(* IEC 61131-3 sources: skladplc/, 9 files *)

(* ---- prgMaindomaci.ST ---- *)
VAR_GLOBAL
cidloAnalog0 at %XW34:int;
cidloAnalog1 at %XW46:int;
cidlo_horiz at %X100.4:bool;
cidlo_verti at %X100.7:bool;
cidlo_rameno_zadni at %X10.7:bool;
doprav_cidlo_zad at %X100.6:bool;
doprav_cidlo_pre at %X100.5:bool;
zk0 at %X101.0:bool;
zk1 at %X101.1:bool;
zk2 at %X101.2:bool;
zk3 at %X101.3:bool;
doprav_do at %Y32.4:bool;//dopravnik, dovnitr
doprav_ve at %Y32.5:bool;//dopravnik, ven
horiz_vl at %Y32.6:bool;//horizontalni, vlevo:ccw
horiz_vp at %Y32.7:bool;//horizontalni, vpravo:cw
verti_do at %Y33.0:bool;//vertikalni, dolu
verti_na at %Y33.1:bool;//vertikalni, nahoru
ram_vy at %Y33.2:bool;//rameno, vysun
ram_vs at %Y33.3:bool;//rameno, vsun
horiz_ink:udint;
verti_ink:udint;
cas at %S13.2:bool;
kalibruj:bool:=0;
misto:bool:=0;

pomoc, pomoc1:bool;

casovac, casovac1, casovac2:TON;
(*
PolohaVerti: array[0..4] of udint :=[3852,1892,204,3420];
PolohaHoriz: array[0..4] of udint:=[9403,6462,3629,12];
Obsazenost: array [0..9] of int:=[0,0,0,0,0,0,0,0,0,0]; //not completed
*)
bar:int;
umistit:bool:=0;
nalozeno:bool:=0;
pozice0:int:=0;
pozice1:int:=0;
pozice2:int:=0;

END_VAR
FUNCTION manualni:bool     //HOTOVO, funkce pro servisni ovladani jednotky, pozdeji se smaze
   horiz_vp:=zk0 and not zk3;
   verti_na:=zk1 and not zk3;
   ram_vs:=zk2 and not zk3;
   horiz_vl:=zk0 and  zk3;
   verti_do:=zk1 and  zk3;
   ram_vy:=zk2 and  zk3;
END_FUNCTION
FUNCTION kalibrace:bool  //HOTOVO, funkce na uvodni kalibraci jednotky
   IF not cidlo_rameno_zadni then;
      ram_vs:=1;
      else ram_vs:=0;
      IF not cidlo_horiz then;
         horiz_vp:=1;
         else horiz_vp:=0;
      END_IF;
      IF not cidlo_verti then;
         verti_na:=1;
         else verti_na:=0;
      END_IF;
   END_IF;
   IF cidlo_rameno_zadni AND cidlo_horiz AND cidlo_verti then;
      kalibrace:=1;
   END_IF;
END_FUNCTION

FUNCTION umisti:bool
   IF cidloAnalog0<cidloAnalog1 then;
      IF verti_ink < 1892 then;
         verti_do:=1;
      ELSE
         verti_do:=0;
      END_IF;
      IF horiz_ink < 6462 then;
         horiz_vl:=1;
      ELSE
         horiz_vl:=0;
      END_IF;
      Obsazenost[pozice1]:=1;

      //
   ELSIF (cidloAnalog0<3600 AND cidloAnalog1<3600) then;
      IF verti_ink < 3852 then;
         verti_do:=1;
      ELSE
         verti_do:=0;
      END_IF;
      IF horiz_ink < 9403 then;
         horiz_vl:=1;
      ELSE
         horiz_vl:=0;
      END_IF;
      Obsazenost[pozice0]:=1;

      //
   ELSIF cidloAnalog0>cidloAnalog1  then;  //
      IF verti_ink < 204 then;
         verti_do:=1;
      ELSE
         verti_do:=0;
      END_IF;
      IF horiz_ink < 3629 then;
         horiz_vl:=1;
      ELSE
         horiz_vl:=0;
      END_IF;
      Obsazenost[pozice2]:=1;

      //
   END_IF;
END_FUNCTION
FUNCTION nakladani:bool //funkce pro posun dopravniku s obrokem do nakladaci oblasti
   IF verti_ink < 3350 then; //dojede na vertikalni polohu nakladaci oblasti
      verti_do:=1;
   ELSE
      verti_do:=0;
      pomoc1:=1;
   END_IF;
   IF horiz_ink < 10 then; //dojede na horizontalni polohu nakladaci oblasti
      horiz_vl:=1;
   ELSE
      horiz_vl:=0;
   END_IF;
   IF pomoc1 and not casovac1.Q then; //pokud je ve vertikalni poloze oblasti, zacne na 3s vysouvat rameno = paleta se posadi na dopravnik v nakl. obasti
      ram_vy:=1;
      casovac1(IN:=1, PT:=T#3s); //misto jednicky promenna - nulovani
   ELSIF nalozeno and casovac1.Q then; //pokud uzivatel stiskne tlacitko, ze barevny obrok vlozil, tak se paleta vrati zpet na rameno a to se zatahne
      doprav_
      ram_vy:=0;
      casovac2(IN:1, PT:=T#3s);
      ram_vs:=ram_vs and casovac2.Q
   END_IF;
END_FUNCTION
FUNCTION barva:int //funkce pro určení barvy + vypsání požadované barvy obroku na displej PLC
//hodnota 31500 pro analogove cidlo znamena, ze na dane pozici je cerna barva = neni bily prouzek
   IF not doprav_cidlo_pre AND doprav_cidlo_zad then;
      doprav_do:=1;

      barva:=-1;
      IF (cidloAnalog0=31500 AND cidloAnalog0>cidloAnalog1) then; //bily obrok, nahore bila
        //vypsat na displej BILA

      ELSIF (cidloAnalog1=31500 AND cidloAnalog0<cidloAnalog1) then; //cerveny obrok, dole bila
        //vypsat na displej CERVENA

      ELSIF (cidloAnalog0=31500 AND cidloAnalog0=cidloAnalog1) then; //modry obrok, nikde bila
        //vypsat na displej MODRA

      END_IF;

   END_IF;
   doprav_do:=doprav_cidlo_zad AND doprav_do;

END_FUNCTION
FUNCTION hybej:bool //funkce, ktera podle definovani barvy z funkce barva() urci na jakou pozici se ma naplnena paleta umistit v regalu
   IF not doprav_cidlo_pre AND doprav_cidlo_zad then;
      doprav_do:=1;
      //sken barvy
      IF (umistit) then;
         IF not doprav_cidlo_zad then; //zajisti, ze dopravnik prestane presouvat prazdnou paletu do zadni oblasti jakmile do ni dorazi
            doprav_do:=1;
            doprav_ve:=doprav_cidlo_pre AND doprav_ve;
            nakladej:=nakladani();
            IF nakladej then;
               umisti();
            END_IF;
         END_IF;
         IF (barva() = 0) then;

         ELSIF (barva() = 1) then;S

         ELSIF (barva () = 2) then;

         END_IF;
      END_IF;
      //ceka na potvrzeni vlozeni - stisk tlacitka
   END_IF;

   doprav_do:=doprav_cidlo_zad AND doprav_do;
END_FUNCTION

PROGRAM prgMain
VAR
   cidlo0, cidlo1:INT;
   pomoc:bool;
END_VAR
horiz_ink:=inkrementalni_horiz;
verti_ink:=inkrementalni_verti;
pomoc:=0;
cidlo0:=cidloAnalog0;
cidlo1:=cidloAnalog1;
IF not kalibruj then;     //uvodni kalibrace a pak uvolni system pro dalsi pouziti
   kalibruj:=kalibrace(); //funkce na uvodni kalibraci jednotky
ELSE
   IF casovac.Q then;
      ridSlovo:=1;
      ridSlovo1:=1;
      pomoc:=1;
      //manualni();
      //hybej();
      barva();
   ELSE
      ridSlovo:=2;
      ridSlovo1:=2;
      casovac(IN:=1, PT:=T#1s);
   END_IF;
END_IF;
END_PROGRAM

(* ---- ridici().ST ---- *)
VAR_GLOBAL
   horizontal:int:=0;
   vertikal:int:=0;
   blokace:bool:=0;
END_VAR
FUNCTION ridici:bool
   IF not blokace then
      IF not nabirani.probehlo then
         nabirani(i:=vertikal, j:=horizontal);
      ELSE
         IF not hybej.odvezl then
            hybej();
         ELSE
            IF not vraceni.vraceno then
               //hlavni_barva:=3;
               vraceni(i:=vertikal, j:=horizontal);
            ELSE
               IF horizontal<2 then //podminka pro posun v polich
                  horizontal:=horizontal+1; //posun v horizontalnim poli
                  nabirani.probehlo:=0;
                  hybej.odvezl:=0;
                  vraceni.vraceno:=0;
               END_IF;
               IF horizontal=2 AND vraceni.vraceno then
                  IF vertikal<2 then
                     vertikal:=vertikal+1;
                     horizontal:=-1;
                  ELSE
                     blokace:=1;
                  END_IF;
               END_IF;
            END_IF;
         END_IF;
      END_IF;
   ELSE
      kalibrace();
   END_IF;
END_FUNCTION

(* ---- kalibrace().ST ---- *)
FUNCTION kalibrace:bool //funkce na kalibraci jednotky
   IF not cidlo_rameno_zad then //zatahne rameno
      ram_vs:=1;
   ELSE
      ram_vs:=0;
      IF not cidlo_horiz then //narazi na horizontalni snimac
         horiz_vp:=1;
      ELSE
         horiz_vp:=0;
      END_IF;
      IF not cidlo_verti then //narazi na vertikalni snimac
         verti_na:=1;
      ELSE
         verti_na:=0;
      END_IF;
   END_IF;
   IF cidlo_rameno_zad AND cidlo_horiz AND cidlo_verti then //"vrati", ze probehla funkce
      kalibrace:=1;
   END_IF;
END_FUNCTION

(* ---- nakladani().st ---- *)
FUNCTION nakladani:bool //funkce pro posun jiz nalozene prazdne palety do dopravnikove oblasti + odebrani naplnene palety
   VAR
      verti:udint:=verti_ink;
      horiz:udint:=horiz_ink;
      pomoc:bool:=0;
      pomoc1:bool:=0;
   END_VAR
   IF verti < 3250 then; //dojede na vertikalni polohu nakladaci oblasti
      verti_do:=1;
   ELSIF verti > 3250 then;
      verti_na:=1;
   ELSE
      verti_do:=0;
      verti_na:=0;
      pomoc1:=1;
   END_IF;
   IF horiz < 10 then; //dojede na horizontalni polohu nakladaci oblasti
      horiz_vl:=1;
   ELSIF horiz > 10 then;
      horiz_vp:=1;
   ELSE
      horiz_vl:=0;
      horiz_vp:=0;
      pomoc:=1;
   END_IF;
   ram_vy:=not cidlo_rameno_pre and pomoc and pomoc1; //pokud je v poloze oblasti, zacne se vysouvat rameno = paleta se posadi na dopravnik v nakl. obasti
   IF nalozeno then; //pokud uzivatel stiskne tlacitko, ze barevny obrok vlozil, tak se paleta vrati zpet na rameno a to se zatahne
      IF verti_ink<3150 then; //vylozi paletu na dopravnik
         verti_na:=1;
      ELSE
         verti_na:=0;
      END_IF;
      //doprav_ve:=1;
      //casovac2(IN:=1, PT:=T#3s);
      //doprav_ve:=not casovac2.Q;
      doprav_ve:=not cidlo_rameno_zad;
      IF verti_ink<3250 then;
         verti_na:=1;
      ELSE
         verti_na:=0;
      END_IF;
      //IF doprav_cidlo_pre and not doprav_cidlo_zad then;
         //casovac2(IN:=0, PT:=T#3s);
         ram_vs:=not cidlo_rameno_zad;
      //END_IF;
   END_IF;
END_FUNCTION

(* ---- barva_FCB.ST ---- *)
FUNCTION_BLOCK barva_FCB //FCB na poznavani barevneho kodovani na boku palet
   VAR_INPUT
      a0:int;
      a1:int;
   END_VAR
   VAR
      h:int:=6; //buffer pro color
   END_VAR
   VAR_OUTPUT
      color:int:=6;
   END_VAR
   IF (h=2 or h=6) and (a0>=5000 or a1>=5000) then //neco vjelo
      IF a0<5000 then //bily pruh dole, CERVENA
         h:=0;
      ELSIF a1<5000 then //bily pruh nahore, MODRA
         h:=1;
      ELSE //zadny bily pruh, BILA
         h:=2;
      END_IF;
   END_IF;
   IF not h=6 AND a0<5000 AND a1<5000 then //ochrana proti falesnym skenum
      color:=h;
      h:=6;
   END_IF;
   IF hybej.odvezl then
      color:=6;
   END_IF;
END_FUNCTION_BLOCK
VAR_GLOBAL
   barva:barva_FCB;
END_VAR

(* ---- hybej_FCB.ST ---- *)
FUNCTION_BLOCK hybej_FCB //funkce pro rozvoz palet
   VAR_INPUT
   END_VAR
   VAR
      vertikalne:bool:=0;
      horizontalne:bool:=0;
      zmacknute:bool:=0;
      plna:bool:=0;
      dole:bool:=0;
      nahore:bool:=0;
   END_VAR
   VAR_OUTPUT
      odvezl:bool:=0;
   END_VAR
   IF not zmacknute then
      IF verti_ink<3350 AND not nahore then //dojede na vertikalni polohu nakladaci oblasti smerem dolu
         verti_do:=1;
         dole:=1;
      ELSIF verti_ink>3350 AND not dole then //dojede na vertikalni polohu nakladaci oblasti smerem nahoru
         verti_na:=1;
         nahore:=1;
      ELSE
         verti_do:=0;
         verti_na:=0;
         vertikalne:=1;
      END_IF;
      IF horiz_ink>75 then //dojede na horizontalni polohu nakladaci oblasti
         horiz_vp:=1;
      ELSE
         horiz_vp:=0;
         horizontalne:=1;
      END_IF;
      ram_vy:=not cidlo_rameno_pre AND vertikalne AND horizontalne; //paleta se posadi na dopravnik v nakl. obasti
      doprav_do:=doprav_cidlo_zad AND not doprav_ve AND vertikalne AND horizontalne; //dopravnik posune paletu dovnitr
      barvuj(a0:=cidloAnalog0,a1:=cidloAnalog1); //sken barvy
      CASE barvuj.color OF //vypise pozadovanou barvu na displej PLC pres PanelMaker
         0:
            hlavni_barva:=0;
         1:
            hlavni_barva:=1;
         2:
            hlavni_barva:=2;
         6:
            hlavni_barva:=3;
      END_CASE;
   END_IF;
   IF nalozeno then //pokud je zmacklo tlacitko, nastavi pomocnou
      zmacknute:=TRUE;
   END_IF;
   IF zmacknute AND not plna then //pokud uzivatel stiskne tlacitko, ze barevny obrok vlozil, tak se paleta vrati zpet na rameno a to se zatahne
      IF verti_ink<3400 then //rameno sjede trochu dolu
         verti_do:=1;
      ELSE
         verti_do:=0;
      END_IF;
   END_IF;
   IF zmacknute AND doprav_cidlo_pre AND not plna then
      doprav_ve:=1;
   ELSIF zmacknute AND not doprav_cidlo_pre AND doprav_cidlo_zad AND not plna then
      doprav_ve:=0;
      plna:=TRUE;
   END_IF;
   IF plna then
      IF verti_ink>3150 then //rameno jiz s paletou vyjede vyse a zatahne se
         verti_na:=1;
      ELSE
         verti_na:=0;
         ram_vs:=not cidlo_rameno_zad;
         odvezl:=cidlo_rameno_zad;
         IF odvezl then //reset vsech pomocnych pro dalsi pouziti
            vertikalne:=0;
            horizontalne:=0;
            zmacknute:=0;
            plna:=0;
            dole:=0;
            nahore:=0;
         END_IF;
      END_IF;
   END_IF;
END_FUNCTION_BLOCK
VAR_GLOBAL
   hybej:hybej_FCB;
END_VAR

(* ---- prgMain.ST ---- *)
VAR_GLOBAL
cidloAnalog0 at %XW34:int; //dolni cidlo na dopravniku - poznava barevny kod na palete
cidloAnalog1 at %XW46:int; //horni cidlo na dopravniku - poznava barevny kod na palete
cidlo_horiz at %X100.4:bool; //mechanicke cidlo na horizontalni ose prepravniku
cidlo_verti at %X100.7:bool; //mechanicke cidlo na vertikalni ose prepravniku
cidlo_rameno_zad at %X10.7:bool; //mechanicke cidlo v zadni casti ramena prepravniku
cidlo_rameno_pre at %X10.6:bool; //mechanicke cidlo v predni casti ramena prepravniku
doprav_cidlo_zad at %X100.6:bool;  //svetelna brana dopravniku vzadu
doprav_cidlo_pre at %X100.5:bool; // svetelna brana dopravniku vpredu
zk0 at %X101.0:bool; //manualni input
zk1 at %X101.1:bool;
zk2 at %X101.2:bool;
zk3 at %X101.3:bool;
doprav_do at %Y32.4:bool; //pohon dopravniku - dovnitr
doprav_ve at %Y32.5:bool; //pohon dopravniku - ven
horiz_vl at %Y32.6:bool; //horizontalni, vlevo:ccw
horiz_vp at %Y32.7:bool; //horizontalni, vpravo:cw
verti_do at %Y33.0:bool; //vertikalni, dolu
verti_na at %Y33.1:bool; //vertikalni, nahoru
ram_vy at %Y33.2:bool; //rameno, vysun
ram_vs at %Y33.3:bool; //rameno, vsun
horiz_ink:udint;
verti_ink:udint;
cas at %S13.2:bool;
kalibruj:bool:=0;
misto:bool:=0;
displejBarva:string;

casovac:TON;

PolohaVerti: array[0..4] of udint:=[3852,1892,204,3420];
PolohaHoriz: array[0..4] of udint:=[9403,6462,3629,12];
Obsazenost:  array[0..9] of int:=[0,0,0,0,0,0,0,0,0,0];

bar:int;
//umistit:bool:=0;
nalozeno:bool:=zk0;

END_VAR
FUNCTION kalibrace:bool  //HOTOVO, funkce na kalibraci jednotky
   IF not cidlo_rameno_zad then;
      ram_vs:=1;
      else ram_vs:=0;
      IF not cidlo_horiz then;
         horiz_vp:=1;
         else horiz_vp:=0;
      END_IF;
      IF not cidlo_verti then;
         verti_na:=1;
         else verti_na:=0;
      END_IF;
   END_IF;
   IF cidlo_rameno_zad AND cidlo_horiz AND cidlo_verti then;
      kalibrace:=1;
   END_IF;
END_FUNCTION
FUNCTION manualni:bool     //HOTOVO, funkce na manualni ovladani
   horiz_vp:=zk0 and not zk3;
   verti_na:=zk1 and not zk3;
   ram_vs:=zk2 and not zk3;
   horiz_vl:=zk0 and  zk3;
   verti_do:=zk1 and  zk3;
   ram_vy:=zk2 and  zk3;
END_FUNCTION
(*
FUNCTION nakladani:bool //funkce pro posun jiz nalozene prazdne palety do dopravnikove oblasti + odebrani naplnene palety
   VAR
      verti:udint:=verti_ink;
      horiz:udint:=horiz_ink;
      pomoc:bool:=0;
      pomoc1:bool:=0;
   END_VAR
   IF verti < 3250 then; //dojede na vertikalni polohu nakladaci oblasti
      verti_do:=1;
   ELSIF verti > 3250 then;
      verti_na:=1;
   ELSE
      verti_do:=0;
      verti_na:=0;
      pomoc1:=1;
   END_IF;
   IF horiz < 10 then; //dojede na horizontalni polohu nakladaci oblasti
      horiz_vl:=1;
   ELSIF horiz > 10 then;
      horiz_vp:=1;
   ELSE
      horiz_vl:=0;
      horiz_vp:=0;
      pomoc:=1;
   END_IF;
   ram_vy:=not cidlo_rameno_pre and pomoc and pomoc1; //pokud je v poloze oblasti, zacne se vysouvat rameno = paleta se posadi na dopravnik v nakl. obasti
   IF nalozeno then; //pokud uzivatel stiskne tlacitko, ze barevny obrok vlozil, tak se paleta vrati zpet na rameno a to se zatahne
      IF verti_ink<3150 then; //vylozi paletu na dopravnik
      	verti_na:=1;
      ELSE
      	verti_na:=0;
      END_IF;
      //doprav_ve:=1;
      //casovac2(IN:=1, PT:=T#3s);
      //doprav_ve:=not casovac2.Q;
      doprav_ve:=not cidlo_rameno_zad;
      IF verti_ink<3250 then;
         verti_na:=1;
      ELSE
         verti_na:=0;
      END_IF;
      //IF doprav_cidlo_pre and not doprav_cidlo_zad then;
         //casovac2(IN:=0, PT:=T#3s);
         ram_vs:=not cidlo_rameno_zad;
      //END_IF;
   END_IF;
END_FUNCTION
*)
FUNCTION_BLOCK color_fb
   var_input
      a0:int;
      a1:int;
   end_var
   var
      h:int:=-1; // buffer pro color
   end_var
   var_output
      color:int:=-1;
   end_var
   if (h=0 or h=-1) and (a0>=5000 or a1>=5000) then;
     // něco vjelo
     if a0<5000 then; //bílý pruh dole
       h:=1;
     elsif a1<5000 then; //bílý pruh nahoře
       h:=2;
     else //žádný bílý pruh
       h:=0;
     end_if;
   end_if;
   if not h=-1 and a0<5000 and a1<5000 then;
     color:=h;
     h:=-1;
   end_if
END_FUNCTION_BLOCK
var_global
   col:color_fb;
   dd:bool:=0;
   done:bool:=0;
end_var

//legacy useless funkce
(*
FUNCTION barva:int  //SKORO, funkce pro určení barvy + vypsání požadované barvy obroku na displej PLC
   barva:=-1;
      IF (cidloAnalog0=31500 AND cidloAnalog0>cidloAnalog1) then; //bila, nahore bila
         //vypsat na displej BILA
         barva:=0;
      ELSIF (cidloAnalog1=31500 AND cidloAnalog0<cidloAnalog1) then; //cervena, dole bila
         //vypsat na displej CERVENA
         barva:=1;
      ELSIF (cidloAnalog0=31500 AND cidloAnalog0=cidloAnalog1) then; //modra, nikde bila
         //vypsat na displej MODRA
         barva:=2;
      END_IF;
END_FUNCTION
*)

FUNCTION hybej:bool //funkce pro rozvoz naplněných palet do regálů
   VAR
      nakladej:bool:=0;
      verti:udint:=verti_ink;
      horiz:udint:=horiz_ink;
      pomoc:bool:=0;
      pomoc1:bool:=0;
			displayInited:=0;
   END_VAR
   IF verti < 3250 then; //dojede na vertikalni polohu nakladaci oblasti
      verti_do:=1;
   ELSIF verti > 3250 then;
      verti_na:=1;
   ELSE
      verti_do:=0;
      verti_na:=0;
      pomoc1:=1;
   END_IF;
   IF horiz < 10 then; //dojede na horizontalni polohu nakladaci oblasti
      horiz_vl:=1;
   ELSIF horiz > 10 then;
      horiz_vp:=1;
   ELSE
      horiz_vl:=0;
      horiz_vp:=0;
      pomoc:=1;
   END_IF;
   ram_vy:=not cidlo_rameno_pre and pomoc and pomoc1; //pokud je v poloze oblasti, zacne se vysouvat rameno = paleta se posadi na dopravnik v nakl. obasti
	 //Adamec je idiot a neumí rozdělit dlouhou funkci do víc funkcí aby to dávalo smysl #1

	 IF not doprav_cidlo_pre AND doprav_cidlo_zad then;
      doprav_do:=1;
      //sken barvy - vypis na obrazovku
			col(a0:=cidloAnalog0,a1:=cidloAnalog1);
			case col.color of
				0:
					displejBarva:="bílá";
				1:
					displajBarva:="červená";
				2:
					displajBarva:="modrá";
			end_case;

      IF nalozeno then; //pokud uzivatel stiskne tlacitko, ze barevny obrok vlozil, tak se paleta vrati zpet na rameno a to se zatahne
         IF verti_ink<3150 then; //vylozi paletu na dopravnik
            verti_na:=1;
         ELSE
            verti_na:=0;
         END_IF;
         //doprav_ve:=1;
         //casovac2(IN:=1, PT:=T#3s);
         //doprav_ve:=not casovac2.Q;
         doprav_ve:= doprav_cidlo_pre;
         IF verti_ink<3250 then;
            verti_na:=1;
         ELSE
            verti_na:=0;
         END_IF;
         IF doprav_cidlo_pre and not doprav_cidlo_zad then;
            casovac2(IN:=0, PT:=T#3s);
            ram_vs:=ram_vs and not casovac2.Q;
         END_IF;
      END_IF;
			elsif displayInited=0 then;
				displajBarva:="neznámá"; //před čtením barvy, nastav výpis na "neznámá"
				displayInited:=1;
   END_IF;	//Adamec je idiot a neumí rozdělit dlouhou funkci do víc funkcí aby to dávalo smysl #2

   //doprav_do:=doprav_cidlo_zad AND doprav_do;
END_FUNCTION
(*
FUNCTION_BLOCK rameno:bool
  var_input
      zvedni:bool;
      poloz:bool;
      verti_ink:udint;
   end_var
   var
      verti:udint:=verti_ink;
      //pomoc:bool:=0;
   end_var
   var_output
      hotovo:bool;
   end_var
   IF zvedni AND not hotovo then;
      IF verti<verti_ink+50 then;
         verti_na:=1;
      ELSE
         verti_na:=0;
      END_IF;
      ram_vs:= not cidlo_rameno_zad;
      IF cidlo_rameno_zad then;
         pomoc:=1;
         hotovo:=1;
      END_IF;
   END_IF;
   IF poloz AND not hotovo then;
      IF verti<verti_ink-50 then;
         verti_do:=1;
      ELSE
         verti_do:=0;
      END_IF;
      ram_vs:= not cidlo_rameno_zad;
      IF cidlo_rameno_zad then;
         pomoc:=1;
         hotovo:=1;
      END_IF;
   END_IF;
END_FUNCTION_BLOCK
*)
FUNCTION_BLOCK prazdne_FCB:bool //FCB pro nabrani prazdnych palet a dovezeni je do nakladaci oblasti
   VAR_INPUT
      i:int;
      j:int;
   END_VAR
   VAR
   (*
      i:int:=0;
      j:int:=0;
      blokace:bool:=0;
   *)
      verti:udint;
   END_VAR
   VAR_OUTPUT
      probehlo:bool:=0;
   END_VAR
   //IF not blokace then;
      IF verti_ink<PolohaVerti[i] then; //posune prepravnik na vertikalni uroven
         verti_do:=1;
      ELSE
         verti_do:=0;
         verti:=verti_ink;
         IF horiz_ink<PolohaHoriz[j] then; //posune prepravnik na horizontalni uroven
            horiz_vl:=1;
         ELSE
            horiz_vl:=0;
            ram_vy:= not cidlo_rameno_pre; //vysune rameno
            IF verti<verti_ink+50 then; //nadzvedne rameno uz s paletou
               verti_na:=1;
            ELSE
               verti_na:=0;
               ram_vs:= not cidlo_rameno_zad; //zasune rameno
            END_IF;
            probehlo:=1;
         END_IF;
      END_IF;
   //END_IF;
END_FUNCTION_BLOCK
VAR_GLOBAL
   nabirani:=prazdne_FCB;
END_VAR
FUNCTION dovez_prazdne:bool
   VAR
      i:int:=0;
      j:int:=0;
      probehlo:bool=0;
      blokace:bool=0;
   END_VAR
   IF probehlo AND not blokace then;
      hybej();
      IF i<=2 AND j<=2 then;
         j:=j+1;
      ELSIF i<2 then;
         i:=i+1;
      ELSE
         blokace:=1;
      END_IF;
   ELSE
      nabirani(i:=i, j:=j, probehlo=>probehlo);
   END_IF;

END_FUNCTION

PROGRAM prgMain
VAR
   cidlo0, cidlo1:INT;
   pomoc:bool;
END_VAR
horiz_ink:=inkrementalni_horiz;
verti_ink:=inkrementalni_verti;
pomoc:=0;
cidlo0:=cidloAnalog0;
cidlo1:=cidloAnalog1;
IF not kalibruj then;     //uvodni kalibrace, zajisti, ze po spusteni se system vzdy nejdrive zkalibruje
   kalibruj:=kalibrace();
ELSE
   IF casovac.Q then; //seridi nejdrive inkrementalni snimace, po te program dale pokracuje
      ridSlovo:=1;
      ridSlovo1:=1;
      pomoc:=1;
      //manualni();
      hybej();
      dovez_prazdne();
   ELSE
      ridSlovo:=2;
      ridSlovo1:=2;
      casovac(IN:=1, PT:=T#1s); //prodleva pro korektni serizeni snimacu
   END_IF;
END_IF;
END_PROGRAM

(* ---- rameno().st ---- *)
FUNCTION_BLOCK rameno:bool
  var_input
      zvedni:bool;
      poloz:bool;
      verti_ink:udint;
   end_var
   var
      verti:udint:=verti_ink;
      //pomoc:bool:=0;
   end_var
   var_output
      hotovo:bool;
   end_var
   IF zvedni AND not hotovo then;
      IF verti<verti_ink+50 then;
         verti_na:=1;
      ELSE
         verti_na:=0;
      END_IF;
      ram_vs:= not cidlo_rameno_zad;
      IF cidlo_rameno_zad then;
         pomoc:=1;
         hotovo:=1;
      END_IF;
   END_IF;
   IF poloz AND not hotovo then;
      IF verti<verti_ink-50 then;
         verti_do:=1;
      ELSE
         verti_do:=0;
      END_IF;
      ram_vs:= not cidlo_rameno_zad;
      IF cidlo_rameno_zad then;
         pomoc:=1;
         hotovo:=1;
      END_IF;
   END_IF;
END_FUNCTION_BLOCK

(* ---- diff.prgMain.ST ---- *)
29,31c29
< casovac, casovac1:TON;
<
<
---
> casovac, casovac1, casovac2:TON;
35c33
< Obsazenost:  array [0..9] of int:=[0,0,0,0,0,0,0,0,0,0];
---
> Obsazenost: array [0..9] of int:=[0,0,0,0,0,0,0,0,0,0]; //not completed
39c37
<
---
> nalozeno:bool:=0;
45c43,51
< FUNCTION kalibrace:bool  //HOTOVO, funkce na kalibraci
---
> FUNCTION manualni:bool     //HOTOVO, funkce pro servisni ovladani jednotky, pozdeji se smaze
>    horiz_vp:=zk0 and not zk3;
>    verti_na:=zk1 and not zk3;
>    ram_vs:=zk2 and not zk3;
>    horiz_vl:=zk0 and  zk3;
>    verti_do:=zk1 and  zk3;
>    ram_vy:=zk2 and  zk3;
> END_FUNCTION
> FUNCTION kalibrace:bool  //HOTOVO, funkce na uvodni kalibraci jednotky
62,70c68,69
< FUNCTION manualni:bool     //HOTOVO, funkce na manualni ovladani pomoci switche
<    horiz_vp:=zk0 and not zk3;
<    verti_na:=zk1 and not zk3;
<    ram_vs:=zk2 and not zk3;
<    horiz_vl:=zk0 and  zk3;
<    verti_do:=zk1 and  zk3;
<    ram_vy:=zk2 and  zk3;
< END_FUNCTION
< FUNCTION umisti:bool       //SKORO, funkce, ktera ma jiz naplnene palety rozmistovat do regalu
---
>
> FUNCTION umisti:bool
82a82
>
114,118c114,115
< FUNCTION nakladani:bool    //DODELAT, funkce pro nosič palet. umístí prázdné palety na přepravník
<    VAR
<       nulovani:int:=1;
<    END_VAR
<    IF verti_ink < 3350 then;
---
> FUNCTION nakladani:bool //funkce pro posun dopravniku s obrokem do nakladaci oblasti
>    IF verti_ink < 3350 then; //dojede na vertikalni polohu nakladaci oblasti
124c121
<    IF horiz_ink < 10 then;
---
>    IF horiz_ink < 10 then; //dojede na horizontalni polohu nakladaci oblasti
129c126
<    IF pomoc1 and not casovac1.Q then;
---
>    IF pomoc1 and not casovac1.Q then; //pokud je ve vertikalni poloze oblasti, zacne na 3s vysouvat rameno = paleta se posadi na dopravnik v nakl. obasti
132,139c129,133
<    ELSIF pomoc1 and casovac1.Q then;
<       nulovani:=1;
<       casovac1(IN:=2, PT:=T#3s);
<       casovac1(IN:=1, PT:=T#3s);
<       IF not casovac1.Q then
<          ram_vy:=0;
<          ram_vs:=1;
<       END_IF;
---
>    ELSIF nalozeno and casovac1.Q then; //pokud uzivatel stiskne tlacitko, ze barevny obrok vlozil, tak se paleta vrati zpet na rameno a to se zatahne
>       doprav_
>       ram_vy:=0;
>       casovac2(IN:1, PT:=T#3s);
>       ram_vs:=ram_vs and casovac2.Q
141a136,139
> FUNCTION barva:int //funkce pro určení barvy + vypsání požadované barvy obroku na displej PLC
> //hodnota 31500 pro analogove cidlo znamena, ze na dane pozici je cerna barva = neni bily prouzek
>    IF not doprav_cidlo_pre AND doprav_cidlo_zad then;
>       doprav_do:=1;
143,188c141,142
< FUNCTION_BLOCK color_fb
<    var_input
<       reset:bool;
<       a0:int;
<       a1:int;
<    end_var
<    var
<       b0:int;
<       b1:int;
<       something:bool;
<    end_var
<    var_output
<       color:int;
<    end_var
<   if reset then;
<     b0:=1;
<     b1:=1;
<     color:=-1;
<     something:=0;
<     reset:=0;
<     else
<       if a0<5000 and b0=1 then;
<          b0:=0;
<       elsif a0>=5000 then;
<          b0:=1;
<          something:=1;
<       end_if;
<       if a1<5000 and b1=1 then;
<          b1:=0;
<       elsif a0>=5000 then;
<          b1:=1;
<          something:=1;
<       end_if;
<       if color=-1 and a0<5000 and a1<5000 and something then;
<          color:=b0+2*b1;
<       end_if;
<   end_if;
< END_FUNCTION_BLOCK
< var_global
< col:color_fb;
< dd:bool:=0;
<       done:bool:=0;
< end_var
< FUNCTION barva:int  //SKORO, funkce pro určení barvy + vypsání požadované barvy obroku na displej PLC
<    barva:=-1;
<       IF (cidloAnalog0=31500 AND cidloAnalog0>cidloAnalog1) then; //bila, nahore bila
---
>       barva:=-1;
>       IF (cidloAnalog0=31500 AND cidloAnalog0>cidloAnalog1) then; //bily obrok, nahore bila
190,191c144,145
<         barva:=0;
<       ELSIF (cidloAnalog1=31500 AND cidloAnalog0<cidloAnalog1) then; //cervena, dole bila
---
>
>       ELSIF (cidloAnalog1=31500 AND cidloAnalog0<cidloAnalog1) then; //cerveny obrok, dole bila
193,194c147,148
<         barva:=1;
<       ELSIF (cidloAnalog0=31500 AND cidloAnalog0=cidloAnalog1) then; //modra, nikde bila
---
>
>       ELSIF (cidloAnalog0=31500 AND cidloAnalog0=cidloAnalog1) then; //modry obrok, nikde bila
196c150
<         barva:=2;
---
>
198c152,155
< END_FUNCTION
---
>
>
>    END_IF;
>    doprav_do:=doprav_cidlo_zad AND doprav_do;
200,203c157,159
< FUNCTION hybej:bool //funkce pro rozvoz naplněných palet do regálů
<    VAR
<       nakladej:bool:=0;
<    END_VAR
---
>
> END_FUNCTION
> FUNCTION hybej:bool //funkce, ktera podle definovani barvy z funkce barva() urci na jakou pozici se ma naplnena paleta umistit v regalu
206,228c162,169
<       //sken barvy - vypis na obrazovku
<       //bar:=barva();
<       if not col.color=-1 then;
<         col(reset:=1);
<       end_if;
<       if col.color=-1 then;
<          col(a0:=cidloAnalog0,a1:=cidloAnalog1);
<          done:=0;
<       else
<          done:=1;
<       end_if;
<       if col.color=1 then;
<          dd:=1;
<       end_if;
<       if not col.color=-1 then;
<          IF (umistit) then;
<             IF not doprav_cidlo_zad then;
<                doprav_ve:=1;
<                doprav_ve:=doprav_cidlo_pre AND doprav_ve;
<                nakladej:=nakladani();
<                IF nakladej then;
<                   umisti();
<                END_IF;
---
>       //sken barvy
>       IF (umistit) then;
>          IF not doprav_cidlo_zad then; //zajisti, ze dopravnik prestane presouvat prazdnou paletu do zadni oblasti jakmile do ni dorazi
>             doprav_do:=1;
>             doprav_ve:=doprav_cidlo_pre AND doprav_ve;
>             nakladej:=nakladani();
>             IF nakladej then;
>                umisti();
230c171,172
<             IF (col.color = 0) then;
---
>          END_IF;
>          IF (barva() = 0) then;
232c174
<             ELSIF (col.color = 1) then;
---
>          ELSIF (barva() = 1) then;S
234c176
<             ELSIF (col.color = 2) then;
---
>          ELSIF (barva () = 2) then;
236d177
<             END_IF;
238c179
<       end_if;
---
>       END_IF;
241,243c182
<    //IF not doprav_cidlo_zad then;
<    //   doprav_do:=0;
<    //END_IF;
---
>
245d183
<
266c204,205
<       hybej();
---
>       //hybej();
>       barva();
268c207
<       ridSlovo:=2;        //serizeni inkrementalnich snimacu
---
>       ridSlovo:=2;
